// TIA Portal V17 export
// export: Created 2024-08-07T21:43:58.8087197Z, ExportSetting WithDefaults, DisplayName Totally Integrated Automation Portal, DisplayVersion V17 Update 7, DisplayName TIA Portal Openness, DisplayVersion V17 Update 7, DisplayName TIA Portal Version Control Interface, DisplayVersion V17, DisplayName SINAMICS Startdrive Advanced, DisplayVersion V17 SP2, DisplayName SINAMICS Startdrive G110M, G120, G120C, G120D, G120P, G115D, DisplayVersion V17 SP2, DisplayName SINAMICS Startdrive G130, G150, S120, S150, SINAMICS MV, S210, DisplayVersion V17 SP2, DisplayName STEP 7 Professional, DisplayVersion V17 Update 7, DisplayName STEP 7 Safety, DisplayVersion V17 Update 6, DisplayName WinCC Advanced / Unified PC, DisplayVersion V17 Update 7
DATA_BLOCK "READER_MODEL_ACTUAL"   // DB75
{ S7_Optimized_Access := 'TRUE' }
VERSION : 0.1
// stored: AutoNumber true, DBAccessibleFromOPCUA true, DBAccessibleFromWebserver true, IsOnlyStoredInLoadMemory false, IsRetainMemResEnabled false, IsWriteProtectedInAS false, MemoryReserve 100
   VAR
      PRODUCTO : "READER_PRODUCT";
      ST1_TABLE_1 : Struct
         SIDE_RH : String;
         SIDE_LH : String;
         REAR_TUBE : String;
         FRONT_TUBE : String;
         NFP_AUX : String;
      END_STRUCT;
      ST2_TABLE_2 : Struct
         SIDE_RH : String;
         SIDE_LH : String;
         REAR_TUBE : String;
         FRONT_TUBE : String;
         NFP_AUX : String;
      END_STRUCT;
      ST3_FITTING : Struct
         SIDE_RH : String;
         SIDE_LH : String;
         REAR_TUBE : String;
         FRONT_TUBE : String;
         NFP_AUX : String;
      END_STRUCT;
      R1_GRIPPER : Struct
         SIDE_RH : String;
         SIDE_LH : String;
         REAR_TUBE : String;
         FRONT_TUBE : String;
         NFP_AUX : String;
      END_STRUCT;
      R2_GRIPPER : Struct
         SIDE_RH : String;
         SIDE_LH : String;
         REAR_TUBE : String;
         FRONT_TUBE : String;
         NFP_AUX : String;
      END_STRUCT;
      ALL_SCANNER_OK : Bool;
      SIDE_LH_SCANNER_OK : Bool;
      SIDE_RH_SCANNER_OK : Bool;
      REAR_TUBE_SCANNER_OK : Bool;
      FRONT_TUBE_SCANNER_OK : Bool;
      IN_BOX : "READER_PRODUCT";
      EDIT : "READER_PRODUCT";
      READER { S7_SetPoint := 'True'} : String;
      ST_CLEAR : Struct
         SIDE_RH : String;
         SIDE_LH : String;
         REAR_TUBE : String;
         FRONT_TUBE : String;
         NFP_AUX : String;
      END_STRUCT;
      SCAN_CLEAR : Bool;
      RECIBIDO_ESCANER_REAR_TUBE : Array[0..254] of Char;
      RECIBIDO_ESCANER_FRONT_TUBE : Array[0..254] of Char;
      RECIBIDO_ESCANER_RH_MEMBER : Array[0..254] of Char;
      RECIBIDO_ESCANER_LH_MEMBER : Array[0..254] of Char;
      RECIBIDO_ESCANER_REAR_TUBE_STRING : String;
      RECIBIDO_ESCANER_FRONT_TUBE_STRING : String;
      RECIBIDO_ESCANER_RH_MEMBER_STRING : String;
      RECIBIDO_ESCANER_LH_MEMBER_STRING : String;
      LECTURA_ESCANER_REAR_TUBE : String;
      LECTURA_ESCANER_FRONT_TUBE : String;
      LECTURA_ESCANER_RH_MEMBER : String;
      LECTURA_ESCANER_LH_MEMBER : String;
   END_VAR
BEGIN
END_DATA_BLOCK
